// TIA Portal V16 export
// export: Created 2023-03-29T11:03:46.3434422Z, ExportSetting WithDefaults, DisplayName Totally Integrated Automation Portal, DisplayVersion V16 Update 6, DisplayName TIA Portal Version Control Interface, DisplayVersion V16 Update 2, DisplayName TIA Portal Openness, DisplayVersion V16 Update 6, DisplayName STEP 7 Professional, DisplayVersion V16 Update 6, DisplayName STEP 7 Safety, DisplayVersion V16, DisplayName WinCC Advanced, DisplayVersion V16 Update 6
VAR_GLOBAL   // PLC tag table "ModbusRTU"
   switch_flow_analog_modbus AT %M79.0 : Bool;   // przełącznik wyboru medium pomiaru przepływu z wy analogowego czy modbus rtu
END_VAR
